SYSTEM simple_project
  (* Version 1.0, 2025-07-09, dakudryashev *)
  APPLICATION simple_projectApp
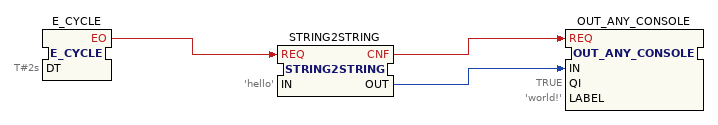
    FBS
      STRING2STRING : STRING2STRING(IN := 'hello');
      E_CYCLE : E_CYCLE(DT := T#2s);
      OUT_ANY_CONSOLE : OUT_ANY_CONSOLE(QI := TRUE, LABEL := 'world!');
    END_FBS
    EVENT_CONNECTIONS
      STRING2STRING.CNF TO OUT_ANY_CONSOLE.REQ;
      E_CYCLE.EO TO STRING2STRING.REQ;
    END_CONNECTIONS
    DATA_CONNECTIONS
      STRING2STRING.OUT TO OUT_ANY_CONSOLE.IN;
    END_CONNECTIONS
  END_APPLICATION
  DEVICE FORTE_PC : FORTE_PC(MGR_ID := "localhost:61499" (* Device manager socket ID *))
    {SET_ATTRIBUTE(Profile, HOLOBLOC)}
    RESOURCE EMB_RES : EMB_RES
      EVENT_CONNECTIONS
        START.COLD TO simple_projectApp.E_CYCLE.START;
        START.WARM TO simple_projectApp.E_CYCLE.START;
      END_CONNECTIONS
    END_RESOURCE
  END_DEVICE
  MAPPINGS
    simple_projectApp.E_CYCLE ON FORTE_PC.EMB_RES;
    simple_projectApp.STRING2STRING ON FORTE_PC.EMB_RES;
    simple_projectApp.OUT_ANY_CONSOLE ON FORTE_PC.EMB_RES;
  END_MAPPINGS
  SEGMENTS
    Ethernet : Ethernet;
  END_SEGMENTS
  LINKS
    FORTE_PC => Ethernet;
  END_LINKS
END_SYSTEM
